Staubli VAL3: MessageHeader.dtx

public num nMagicNumber
public num nProtocolVersion
public num nMsgType
public num nMsgSequenceNumber
public num nPayloadSize
public num nHeaderSize
